// TIA Portal V18 export
FUNCTION_BLOCK "CheckPositioningOrder"   // FB1, LAD
{ S7_Optimized_Access := 'TRUE' }
VERSION : 0.1
// stored: AutoNumber true, IsIECCheckEnabled false, IsRetainMemResEnabled false, MemoryReserve 100, SetENOAutomatically false, UDAEnableTagReadback false
   VAR_INPUT
      "V90Servo[3]" : Struct
         i : Int;
         nError : Int;
         nWarning : Int;
         nPositionListNo : Int := 1;
         Pos : "PosList";
         Point : Array[0..39] of Struct
            Start : Bool;
            Achieve : Bool;
         END_STRUCT;
      END_STRUCT;
   END_VAR
   VAR_OUTPUT
      HaveAxisStart : Bool;
      AxisStartNumber : Int;
   END_VAR
   VAR
      Index : Int;
   END_VAR
BEGIN

REGION Network 2 (SCL)
   FOR #Index := 0 TO 39 DO
       IF #"V90Servo[3]".Point[#Index].Start THEN
           #HaveAxisStart := true;
           #AxisStartNumber := #Index;
           EXIT;
       ELSE
           #HaveAxisStart := FALSE;
           #AxisStartNumber := 32767;
       END_IF;
   END_FOR;
END_REGION
END_FUNCTION_BLOCK
